PROGRAM MAIN
VAR
END_VAR

P_FreeRoom();
P_FreeRoom2();

END_PROGRAM

(* stored: Version 1.1.0.1, ProductVersion 3.1.4024.0
   POU MAIN: Id {5d142a1d-656d-4c31-aef1-167d5220e920}, SpecialFunc None *)
